ABB RobotStudio station: Robot_1200 (task 2).rsstn

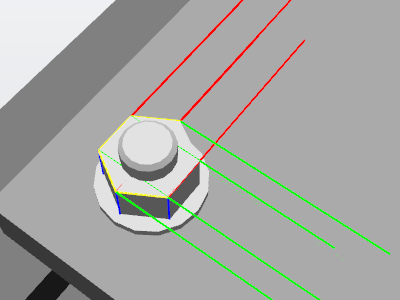
Station Robot_1200 (task 3) @ 7020 (saved by RobotStudio 22.3.10141.1)
Controller Controller18, task T_ROB1: task frame (RAPID world) sits at (0, 0, 290) mm in the station
Controller Controller18
  mechanical unit ROB_1: IRB1200_5_90_STD_03, 6 joints, base frame (0, 0, 0) mm
Layout (positions relative to the parent item):
  - Part_1 [part, from Robotics 7020\Cement Base.rslib] at (-450, -450, 0) mm
  - IRB1200_5_90_STD_03 [mechanism, from %ABB.RobotStudio.Models.IRB1200%\IRB1200_5_90_STD_03.rslib] at (0, 0, 290) mm; joint values [-0.032, 0.8092, 0.5108, -0.033, -1.3351, 0.0082] (rad or m)
  - table_and_fixture_140 [part, from Training Objects\propeller_table.rslib] at (481.47, -175, -3.86) mm
  - Pen_4 [mechanism, from Training Objects\Pen.rslib] at (558.59, -15.28, 573.03) mm, rotated rx 0 ry 89.14 rz 0 deg
Attachment: Pen_4 is attached to IRB1200_5_90_STD_03 / Link6
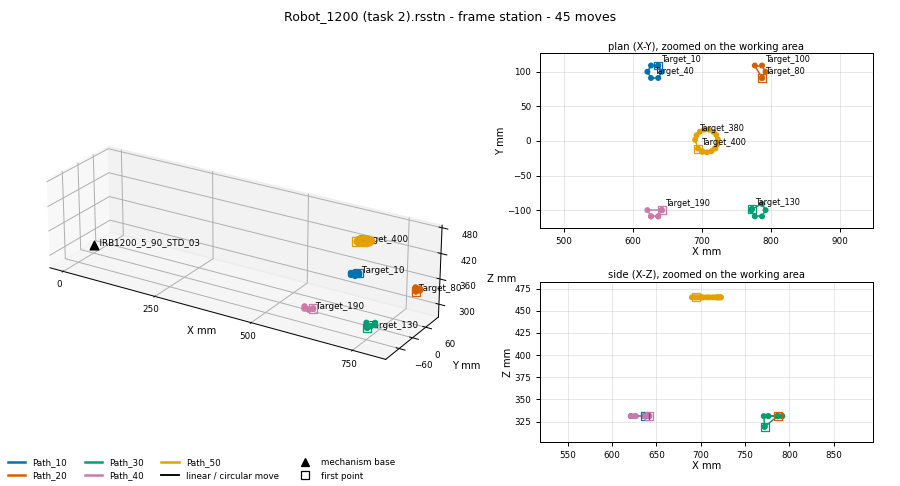
[picture p0: tool path of Robot_1200 (task 2).rsstn in frame station, 45 of 45 moves have a stored position in this frame; points joined in program order, loops and branches not executed]
Targets, tools, work objects and paths stored in the station, written as RAPID:
! task T_ROB1
MODULE CalibData
  PERS tooldata Pen_TCP:=[TRUE,[[110,0,140],[0.707106781,0,0.707106781,0]],[1,[10.7435139,0,140],[1,0,0,0],0,0,0]];
ENDMODULE

! task T_ROB1
MODULE Module1
  CONST robtarget Target_10:=[[636.669544162,108.999991346,41.141031337],[0.007491182,0.000000052,0.999971941,-0.000000029],[0,0,0,1],[9E+09,9E+09,9E+09,9E+09,9E+09,9E+09]];
  CONST robtarget Target_20:=[[626.277290695,108.999981848,41.141021726],[0.007491184,0.000000071,0.999971941,-0.000000035],[0,0,0,1],[9E+09,9E+09,9E+09,9E+09,9E+09,9E+09]];
  CONST robtarget Target_30:=[[621.081106807,99.999997736,41.141069534],[0.007491221,0.000000075,0.99997194,-0.000000031],[0,0,0,1],[9E+09,9E+09,9E+09,9E+09,9E+09,9E+09]];
  CONST robtarget Target_40:=[[626.277320284,90.999992874,41.14107191],[0.007491214,0.000000079,0.99997194,-0.000000027],[0,0,0,1],[9E+09,9E+09,9E+09,9E+09,9E+09,9E+09]];
  CONST robtarget Target_50:=[[636.669542519,90.999996799,41.14103549],[0.007491197,0.000000077,0.999971941,-0.000000025],[0,0,0,1],[9E+09,9E+09,9E+09,9E+09,9E+09,9E+09]];
  CONST robtarget Target_60:=[[641.865647555,99.999993763,41.14104766],[0.007491219,0.000000075,0.99997194,-0.000000029],[0,0,0,1],[9E+09,9E+09,9E+09,9E+09,9E+09,9E+09]];
  CONST robtarget Target_70:=[[636.669553711,108.999991689,41.141058166],[0.007491242,0.000000082,0.99997194,-0.000000024],[0,0,0,1],[9E+09,9E+09,9E+09,9E+09,9E+09,9E+09]];
  CONST robtarget Target_80:=[[786.669580181,90.999998634,41.141033135],[0.007491315,0.000000083,0.99997194,-0.000000018],[0,0,-1,1],[9E+09,9E+09,9E+09,9E+09,9E+09,9E+09]];
  CONST robtarget Target_90:=[[791.865662147,99.99999388,41.141003618],[0.007491284,0.000000095,0.99997194,-0.000000024],[0,0,-1,1],[9E+09,9E+09,9E+09,9E+09,9E+09,9E+09]];
  CONST robtarget Target_100:=[[786.669593225,108.999995295,41.141056614],[0.007491265,0.000000082,0.99997194,-0.000000039],[0,0,-1,1],[9E+09,9E+09,9E+09,9E+09,9E+09,9E+09]];
  CONST robtarget Target_110:=[[776.277168018,108.999999823,41.141063515],[0.007491278,0.00000008,0.99997194,-0.000000037],[0,0,-1,1],[9E+09,9E+09,9E+09,9E+09,9E+09,9E+09]];
  CONST robtarget Target_120:=[[757.977476367,108.999991164,42.451989833],[0.007491347,0.000000079,0.999971939,-0.000000029],[0,0,-1,1],[9E+09,9E+09,9E+09,9E+09,9E+09,9E+09]];
  CONST robtarget Target_130:=[[772.086003325,-98.463207147,29.07515776],[0.007491336,0.000000087,0.99997194,-0.000000035],[-1,-1,0,1],[9E+09,9E+09,9E+09,9E+09,9E+09,9E+09]];
  CONST robtarget Target_140:=[[786.669597862,-90.99999605,41.141074043],[0.007491422,0.000000077,0.999971939,-0.000000043],[-1,-1,0,1],[9E+09,9E+09,9E+09,9E+09,9E+09,9E+09]];
  CONST robtarget Target_150:=[[791.865698469,-100.000005528,41.141087173],[0.007491333,0.00000009,0.99997194,-0.000000031],[-1,-1,0,1],[9E+09,9E+09,9E+09,9E+09,9E+09,9E+09]];
  CONST robtarget Target_160:=[[786.669564812,-108.99999477,41.140998738],[0.007491309,0.000000098,0.99997194,-0.000000025],[-1,-1,0,1],[9E+09,9E+09,9E+09,9E+09,9E+09,9E+09]];
  CONST robtarget Target_170:=[[776.27717009,-108.999995152,41.141073738],[0.007491321,0.000000097,0.99997194,-0.000000019],[-1,-1,0,1],[9E+09,9E+09,9E+09,9E+09,9E+09,9E+09]];
  CONST robtarget Target_180:=[[771.081081569,-100.000002125,41.141081823],[0.007491296,0.000000096,0.99997194,-0.000000017],[-1,-1,0,1],[9E+09,9E+09,9E+09,9E+09,9E+09,9E+09]];
  CONST robtarget Target_190:=[[641.865661601,-100.000002947,41.141066206],[0.007491262,0.000000097,0.99997194,-0.000000019],[-1,-1,-1,1],[9E+09,9E+09,9E+09,9E+09,9E+09,9E+09]];
  CONST robtarget Target_200:=[[636.669540748,-109.000001831,41.141026447],[0.007491287,0.000000113,0.99997194,-0.000000014],[-1,-1,-1,1],[9E+09,9E+09,9E+09,9E+09,9E+09,9E+09]];
  CONST robtarget Target_210:=[[626.277302606,-108.999994181,41.141059424],[0.007491271,0.00000011,0.99997194,-0.000000016],[-1,-1,-1,1],[9E+09,9E+09,9E+09,9E+09,9E+09,9E+09]];
  CONST robtarget Target_220:=[[621.081103143,-99.99999841,41.141051588],[0.007491399,0.000000079,0.999971939,-0.000000023],[-1,-1,-1,1],[9E+09,9E+09,9E+09,9E+09,9E+09,9E+09]];
  CONST robtarget Target_230:=[[626.277314819,-90.999993434,41.141053284],[0.007491393,0.000000074,0.999971939,-0.000000026],[-1,-1,-1,1],[9E+09,9E+09,9E+09,9E+09,9E+09,9E+09]];
  CONST robtarget Target_240:=[[636.66957888,-91.000002762,41.141091367],[0.007491435,0.000000075,0.999971939,-0.000000033],[-1,-1,-1,1],[9E+09,9E+09,9E+09,9E+09,9E+09,9E+09]];
  CONST robtarget Target_250:=[[700.218970713,-15.27686971,175.141107609],[0.007491428,0.000000083,0.999971939,-0.000000033],[-1,-1,0,1],[9E+09,9E+09,9E+09,9E+09,9E+09,9E+09]];
  CONST robtarget Target_260:=[[706.973353828,-16.499998182,175.141092833],[0.007491429,0.000000082,0.999971939,-0.000000033],[-1,-1,0,1],[9E+09,9E+09,9E+09,9E+09,9E+09,9E+09]];
  CONST robtarget Target_270:=[[713.64127001,-14.870130041,175.141099406],[0.007491454,0.000000082,0.999971939,-0.000000033],[-1,-1,0,1],[9E+09,9E+09,9E+09,9E+09,9E+09,9E+09]];
  CONST robtarget Target_280:=[[719.069875663,-10.669079506,175.141099414],[0.007491451,0.000000082,0.999971939,-0.000000033],[-1,-1,0,1],[9E+09,9E+09,9E+09,9E+09,9E+09,9E+09]];
  CONST robtarget Target_290:=[[719.069875663,-10.669079506,175.141099414],[0.007491451,0.000000082,0.999971939,-0.000000033],[-1,-1,0,1],[9E+09,9E+09,9E+09,9E+09,9E+09,9E+09]];
  CONST robtarget Target_300:=[[719.069875663,-10.669079557,175.141099414],[0.007491451,0.000000082,0.999971939,-0.000000033],[-1,-1,0,1],[9E+09,9E+09,9E+09,9E+09,9E+09,9E+09]];
  CONST robtarget Target_310:=[[722.3203603,-4.623251722,175.141091954],[0.007491434,0.000000082,0.999971939,-0.000000033],[-1,-1,0,1],[9E+09,9E+09,9E+09,9E+09,9E+09,9E+09]];
  CONST robtarget Target_320:=[[722.830755069,2.221981052,175.141084556],[0.007491434,0.000000082,0.999971939,-0.000000033],[0,0,-1,1],[9E+09,9E+09,9E+09,9E+09,9E+09,9E+09]];
  CONST robtarget Target_330:=[[720.512786517,8.683012488,175.141082043],[0.007491444,0.000000082,0.999971939,-0.000000034],[0,0,-1,1],[9E+09,9E+09,9E+09,9E+09,9E+09,9E+09]];
  CONST robtarget Target_340:=[[716.57638355,13.054889122,175.141103935],[0.007491439,0.000000082,0.999971939,-0.000000033],[0,0,-1,1],[9E+09,9E+09,9E+09,9E+09,9E+09,9E+09]];
  CONST robtarget Target_350:=[[709.903998297,16.139429343,175.141103664],[0.007491471,0.000000083,0.999971939,-0.000000033],[0,0,-1,1],[9E+09,9E+09,9E+09,9E+09,9E+09,9E+09]];
  CONST robtarget Target_360:=[[703.042897848,16.139430247,175.141103695],[0.007491476,0.000000082,0.999971938,-0.000000033],[0,0,-1,1],[9E+09,9E+09,9E+09,9E+09,9E+09,9E+09]];
  CONST robtarget Target_370:=[[696.774992107,13.348779542,175.141099006],[0.00749149,0.000000082,0.999971938,-0.000000033],[0,0,-1,1],[9E+09,9E+09,9E+09,9E+09,9E+09,9E+09]];
  CONST robtarget Target_380:=[[692.18394931,8.249999711,175.141075813],[0.007491482,0.000000082,0.999971938,-0.000000034],[0,0,-1,1],[9E+09,9E+09,9E+09,9E+09,9E+09,9E+09]];
  CONST robtarget Target_390:=[[690.063742084,1.724719982,175.141083255],[0.007491397,0.000000084,0.999971939,-0.000000029],[0,0,-1,1],[9E+09,9E+09,9E+09,9E+09,9E+09,9E+09]];
  CONST robtarget Target_400:=[[694.211464209,-11.040649535,175.14110766],[0.007491376,0.000000084,0.999971939,-0.000000029],[-1,-1,0,1],[9E+09,9E+09,9E+09,9E+09,9E+09,9E+09]];
  CONST robtarget Target_410:=[[588.25763964,0,682.837205584],[0.258819045,0,-0.965925826,0],[0,0,0,0],[9E+09,9E+09,9E+09,9E+09,9E+09,9E+09]];
  CONST robtarget Target_190_3:=[[641.865661601,-100.000002947,41.141066206],[0.007491262,0.000000097,0.99997194,-0.000000019],[-1,-1,-1,1],[9E+09,9E+09,9E+09,9E+09,9E+09,9E+09]];
  CONST robtarget Target_200_3:=[[636.669540748,-109.000001831,41.141026447],[0.007491287,0.000000113,0.99997194,-0.000000014],[-1,-1,-1,1],[9E+09,9E+09,9E+09,9E+09,9E+09,9E+09]];
  CONST robtarget Target_210_3:=[[626.277302606,-108.999994181,41.141059424],[0.007491271,0.00000011,0.99997194,-0.000000016],[-1,-1,-1,1],[9E+09,9E+09,9E+09,9E+09,9E+09,9E+09]];
  CONST robtarget Target_220_2:=[[621.081103143,-99.99999841,41.141051588],[0.007491399,0.000000079,0.999971939,-0.000000023],[-1,-1,-1,1],[9E+09,9E+09,9E+09,9E+09,9E+09,9E+09]];
  CONST robtarget Target_230_2:=[[626.277314819,-90.999993434,41.141053284],[0.007491393,0.000000074,0.999971939,-0.000000026],[-1,-1,-1,1],[9E+09,9E+09,9E+09,9E+09,9E+09,9E+09]];
  CONST robtarget Target_240_2:=[[636.66957888,-91.000002762,41.141091367],[0.007491435,0.000000075,0.999971939,-0.000000033],[-1,-1,-1,1],[9E+09,9E+09,9E+09,9E+09,9E+09,9E+09]];
  CONST robtarget Target_250_2:=[[700.218970713,-15.27686971,175.141107609],[0.007491428,0.000000083,0.999971939,-0.000000033],[-1,-1,0,1],[9E+09,9E+09,9E+09,9E+09,9E+09,9E+09]];
  CONST robtarget Target_420:=[[700.219008234,-15.276868517,175.141084046],[0.007491398,0.000000082,0.999971939,-0.000000032],[-1,-1,0,1],[9E+09,9E+09,9E+09,9E+09,9E+09,9E+09]];
  PROC Path_10()
    MoveL Target_10,v1000,fine,Pen_TCP\WObj:=wobj0;
    MoveL Target_20,v1000,fine,Pen_TCP\WObj:=wobj0;
    MoveL Target_30,v1000,fine,Pen_TCP\WObj:=wobj0;
    MoveL Target_40,v1000,fine,Pen_TCP\WObj:=wobj0;
    MoveL Target_50,v1000,fine,Pen_TCP\WObj:=wobj0;
    MoveL Target_60,v1000,fine,Pen_TCP\WObj:=wobj0;
    MoveL Target_10,v1000,fine,Pen_TCP\WObj:=wobj0;
  ENDPROC
  PROC Path_20()
    MoveL Target_80,v1000,fine,Pen_TCP\WObj:=wobj0;
    MoveL Target_90,v1000,fine,Pen_TCP\WObj:=wobj0;
    MoveL Target_100,v1000,fine,Pen_TCP\WObj:=wobj0;
    MoveL Target_110,v1000,fine,Pen_TCP\WObj:=wobj0;
    MoveL Target_80,v1000,fine,Pen_TCP\WObj:=wobj0;
  ENDPROC
  PROC Path_30()
    MoveL Target_130,v1000,fine,Pen_TCP\WObj:=wobj0;
    MoveL Target_140,v1000,fine,Pen_TCP\WObj:=wobj0;
    MoveL Target_150,v1000,fine,Pen_TCP\WObj:=wobj0;
    MoveL Target_160,v1000,fine,Pen_TCP\WObj:=wobj0;
    MoveL Target_170,v1000,fine,Pen_TCP\WObj:=wobj0;
    MoveL Target_180,v1000,fine,Pen_TCP\WObj:=wobj0;
    MoveL Target_130,v1000,fine,Pen_TCP\WObj:=wobj0;
  ENDPROC
  PROC Path_40()
    MoveL Target_190,v80,fine,Pen_TCP\WObj:=wobj0;
    MoveL Target_190_3,v80,fine,Pen_TCP\WObj:=wobj0;
    MoveL Target_200,v80,fine,Pen_TCP\WObj:=wobj0;
    MoveL Target_200_3,v80,fine,Pen_TCP\WObj:=wobj0;
    MoveL Target_210,v80,fine,Pen_TCP\WObj:=wobj0;
    MoveL Target_210_3,v80,fine,Pen_TCP\WObj:=wobj0;
    MoveL Target_220,v80,fine,Pen_TCP\WObj:=wobj0;
    MoveL Target_190,v80,fine,Pen_TCP\WObj:=wobj0;
  ENDPROC
  PROC Path_50()
    MoveL Target_400,v80,fine,Pen_TCP\WObj:=wobj0;
    MoveL Target_390,v80,fine,Pen_TCP\WObj:=wobj0;
    MoveL Target_380,v80,fine,Pen_TCP\WObj:=wobj0;
    MoveL Target_370,v80,fine,Pen_TCP\WObj:=wobj0;
    MoveL Target_360,v80,fine,Pen_TCP\WObj:=wobj0;
    MoveL Target_350,v80,fine,Pen_TCP\WObj:=wobj0;
    MoveL Target_340,v80,fine,Pen_TCP\WObj:=wobj0;
    MoveL Target_330,v80,fine,Pen_TCP\WObj:=wobj0;
    MoveL Target_320,v80,fine,Pen_TCP\WObj:=wobj0;
    MoveL Target_310,v80,fine,Pen_TCP\WObj:=wobj0;
    MoveL Target_300,v80,fine,Pen_TCP\WObj:=wobj0;
    MoveL Target_290,v80,fine,Pen_TCP\WObj:=wobj0;
    MoveL Target_280,v80,fine,Pen_TCP\WObj:=wobj0;
    MoveL Target_270,v80,fine,Pen_TCP\WObj:=wobj0;
    MoveL Target_260,v80,fine,Pen_TCP\WObj:=wobj0;
    MoveL Target_250_2,v80,fine,Pen_TCP\WObj:=wobj0;
    MoveL Target_250,v80,fine,Pen_TCP\WObj:=wobj0;
    MoveL Target_250,v80,fine,Pen_TCP\WObj:=wobj0;
  ENDPROC
ENDMODULE

